(* CODESYS project lab3_pod2.project
   Title: lab2_pod2
   Version: 0.0.0.0
   Author: ichiro

Project tree, tasks and I/O mapping:
  MyController : TM251MESE, Schneider Electric, order no. TM251MESE, version 4.0.6.18
    application Application
      task MAST (cyclic, interval t#1s, priority 15, watchdog 100 ms x 1) calls Task1_1
      global variables GVL
      program TASK1 [ST]
      program TASK2 [ST]
      program TASK3 [ST]
      program TASK5 [ST]
      program TASK4 [ST]
      program Task1_1 [ST]
      Relocation Table
    IO_Bus : IO bus - TM3, Schneider Electric, version 4.0.6.18
      Module_1 : TM3TM3/G, Schneider Electric, order no. TM3TM3/G, version 1.0.1.6
          settings: KPI Configuration.KPI Configuration[0] = 78; KPI Configuration.KPI Configuration[1] = 35; KPI Configuration.KPI Configuration[2] = 48; KPI Configuration.KPI Configuration[3] = 248; KPI Configuration.KPI Configuration[5] = 0; KPI Configuration.KPI Configuration[6] = 112; KPI Configuration.KPI Configuration[7] = 23; KPI Configuration.KPI Configuration[8] = 100; KPI Configuration.KPI Configuration[9] = 0; KPI Configuration.KPI Configuration[16] = 16; KPI Configuration.KPI Configuration[19] = 0; KPI Configuration.KPI Configuration[20] = 192; KPI Configuration.KPI Configuration[21] = 93
          input  temper_in : INT  // IW0
          input  water_in : INT  // IW1
          output motor : INT  // QW0
          input  ibModule_1_IBStatusIW0 : BYTE  // IBStatusIW0
          input  ibModule_1_IBStatusIW1 : BYTE  // IBStatusIW1
          input  ibModule_1_IBStatusQW0 : BYTE  // IBStatusQW0
    COM_Bus : COM bus, Schneider Electric, version 4.0.6.18
    Ethernet_1 : Ethernet Network, Schneider Electric, version 4.0.6.18
      ModbusTCP_Slave_Device : ModbusTCP Slave Device, Schneider Electric, version 3.5.2.6
          input  iwModbusTCP_Slave_Device_Inputs_0 : WORD  // Inputs.Inputs[0]
          input  iwModbusTCP_Slave_Device_Inputs_1 : WORD  // Inputs.Inputs[1]
          input  iwModbusTCP_Slave_Device_Inputs_2 : WORD  // Inputs.Inputs[2]
          input  iwModbusTCP_Slave_Device_Inputs_3 : WORD  // Inputs.Inputs[3]
          input  iwModbusTCP_Slave_Device_Inputs_4 : WORD  // Inputs.Inputs[4]
          input  iwModbusTCP_Slave_Device_Inputs_5 : WORD  // Inputs.Inputs[5]
          input  iwModbusTCP_Slave_Device_Inputs_6 : WORD  // Inputs.Inputs[6]
          input  iwModbusTCP_Slave_Device_Inputs_7 : WORD  // Inputs.Inputs[7]
          input  iwModbusTCP_Slave_Device_Inputs_8 : WORD  // Inputs.Inputs[8]
          input  iwModbusTCP_Slave_Device_Inputs_9 : WORD  // Inputs.Inputs[9]
          output qwModbusTCP_Slave_Device_Outputs_0 : WORD  // Outputs.Outputs[0]
          output qwModbusTCP_Slave_Device_Outputs_1 : WORD  // Outputs.Outputs[1]
          output qwModbusTCP_Slave_Device_Outputs_2 : WORD  // Outputs.Outputs[2]
          output qwModbusTCP_Slave_Device_Outputs_3 : WORD  // Outputs.Outputs[3]
          output qwModbusTCP_Slave_Device_Outputs_4 : WORD  // Outputs.Outputs[4]
          output qwModbusTCP_Slave_Device_Outputs_5 : WORD  // Outputs.Outputs[5]
          output qwModbusTCP_Slave_Device_Outputs_6 : WORD  // Outputs.Outputs[6]
          output qwModbusTCP_Slave_Device_Outputs_7 : WORD  // Outputs.Outputs[7]
          output qwModbusTCP_Slave_Device_Outputs_8 : WORD  // Outputs.Outputs[8]
          output qwModbusTCP_Slave_Device_Outputs_9 : WORD  // Outputs.Outputs[9]
          unmapped channels: Inputs, Outputs
    Ethernet_2 : Device Network, Schneider Electric, version 4.0.6.18
        settings: IPAddress = [10, 77, 70, 112]; SubnetMask = [255, 255, 255, 0]; GatewayAddress = [10, 77, 70, 1]; WebServer = TRUE; FTP Server = TRUE; SoMachine Protocol = TRUE; Modbus Server = TRUE; NetManage Protocol = TRUE; SNMP protocol = TRUE; Enable Routing = FALSE; WebVisu protocol = TRUE; DHCP Server Active = TRUE
      Industrial_Ethernet_Manager : Industrial Ethernet Manager, Schneider Electric, version 1.0.12.20
          settings: BinaryFileSize = 396; Dhcps Host 0.Client Mac Address = [16#0, 16#0, 16#0, 16#0, 16#0]; Dhcps Host 0.Client Device Name = 'DEVICE_1'; Dhcps Host 0.Client IP Address = [10, 77, 70, 111]; Dhcps Host 0.Network Mask = [255, 255, 255, 0]; Dhcps Host 0.Default Gateway = [10, 77, 70, 112]; Dhcps Host 1.Client Mac Address = [16#0, 16#0, 16#0, 16#0, 16#0]; Dhcps Host 2.Client Mac Address = [16#0, 16#0, 16#0, 16#0, 16#0]; Dhcps Host 3.Client Mac Address = [16#0, 16#0, 16#0, 16#0, 16#0]; Dhcps Host 4.Client Mac Address = [16#0, 16#0, 16#0, 16#0, 16#0]; Dhcps Host 5.Client Mac Address = [16#0, 16#0, 16#0, 16#0, 16#0]; Dhcps Host 6.Client Mac Address = [16#0, 16#0, 16#0, 16#0, 16#0]; Dhcps Host 7.Client Mac Address = [16#0, 16#0, 16#0, 16#0, 16#0]; Dhcps Host 8.Client Mac Address = [16#0, 16#0, 16#0, 16#0, 16#0]; Dhcps Host 9.Client Mac Address = [16#0, 16#0, 16#0, 16#0, 16#0]; Dhcps Host 10.Client Mac Address = [16#0, 16#0, 16#0, 16#0, 16#0]; Dhcps Host 11.Client Mac Address = [16#0, 16#0, 16#0, 16#0, 16#0]; Dhcps Host 12.Client Mac Address = [16#0, 16#0, 16#0, 16#0, 16#0]; Dhcps Host 13.Client Mac Address = [16#0, 16#0, 16#0, 16#0, 16#0]; Dhcps Host 14.Client Mac Address = [16#0, 16#0, 16#0, 16#0, 16#0]; Dhcps Host 15.Client Mac Address = [16#0, 16#0, 16#0, 16#0, 16#0]; Dhcps Host 16.Client Mac Address = [16#0, 16#0, 16#0, 16#0, 16#0]; Dhcps Host 17.Client Mac Address = [16#0, 16#0, 16#0, 16#0, 16#0]; Dhcps Host 18.Client Mac Address = [16#0, 16#0, 16#0, 16#0, 16#0]; Dhcps Host 19.Client Mac Address = [16#0, 16#0, 16#0, 16#0, 16#0]; Dhcps Host 20.Client Mac Address = [16#0, 16#0, 16#0, 16#0, 16#0]; Dhcps Host 21.Client Mac Address = [16#0, 16#0, 16#0, 16#0, 16#0]; Dhcps Host 22.Client Mac Address = [16#0, 16#0, 16#0, 16#0, 16#0]; Dhcps Host 23.Client Mac Address = [16#0, 16#0, 16#0, 16#0, 16#0]; Dhcps Host 24.Client Mac Address = [16#0, 16#0, 16#0, 16#0, 16#0]; Dhcps Host 25.Client Mac Address = [16#0, 16#0, 16#0, 16#0, 16#0]; Dhcps Host 26.Client Mac Address = [16#0, 16#0, 16#0, 16#0, 16#0]; Dhcps Host 27.Client Mac Address = [16#0, 16#0, 16#0, 16#0, 16#0]; Dhcps Host 28.Client Mac Address = [16#0, 16#0, 16#0, 16#0, 16#0]; Dhcps Host 29.Client Mac Address = [16#0, 16#0, 16#0, 16#0, 16#0]; Dhcps Host 30.Client Mac Address = [16#0, 16#0, 16#0, 16#0, 16#0]; Dhcps Host 31.Client Mac Address = [16#0, 16#0, 16#0, 16#0, 16#0]; Dhcps Host 32.Client Mac Address = [16#0, 16#0, 16#0, 16#0, 16#0]; Dhcps Host 33.Client Mac Address = [16#0, 16#0, 16#0, 16#0, 16#0]; Dhcps Host 34.Client Mac Address = [16#0, 16#0, 16#0, 16#0, 16#0];
            Dhcps Host 35.Client Mac Address = [16#0, 16#0, 16#0, 16#0, 16#0]; Dhcps Host 36.Client Mac Address = [16#0, 16#0, 16#0, 16#0, 16#0]; Dhcps Host 37.Client Mac Address = [16#0, 16#0, 16#0, 16#0, 16#0]; Dhcps Host 38.Client Mac Address = [16#0, 16#0, 16#0, 16#0, 16#0]; Dhcps Host 39.Client Mac Address = [16#0, 16#0, 16#0, 16#0, 16#0]; Dhcps Host 40.Client Mac Address = [16#0, 16#0, 16#0, 16#0, 16#0]; Dhcps Host 41.Client Mac Address = [16#0, 16#0, 16#0, 16#0, 16#0]; Dhcps Host 42.Client Mac Address = [16#0, 16#0, 16#0, 16#0, 16#0]; Dhcps Host 43.Client Mac Address = [16#0, 16#0, 16#0, 16#0, 16#0]; Dhcps Host 44.Client Mac Address = [16#0, 16#0, 16#0, 16#0, 16#0]; Dhcps Host 45.Client Mac Address = [16#0, 16#0, 16#0, 16#0, 16#0]; Dhcps Host 46.Client Mac Address = [16#0, 16#0, 16#0, 16#0, 16#0]; Dhcps Host 47.Client Mac Address = [16#0, 16#0, 16#0, 16#0, 16#0]; Dhcps Host 48.Client Mac Address = [16#0, 16#0, 16#0, 16#0, 16#0]; Dhcps Host 49.Client Mac Address = [16#0, 16#0, 16#0, 16#0, 16#0]; Dhcps Host 50.Client Mac Address = [16#0, 16#0, 16#0, 16#0, 16#0]; Dhcps Host 51.Client Mac Address = [16#0, 16#0, 16#0, 16#0, 16#0]; Dhcps Host 52.Client Mac Address = [16#0, 16#0, 16#0, 16#0, 16#0]; Dhcps Host 53.Client Mac Address = [16#0, 16#0, 16#0, 16#0, 16#0]; Dhcps Host 54.Client Mac Address = [16#0, 16#0, 16#0, 16#0, 16#0]; Dhcps Host 55.Client Mac Address = [16#0, 16#0, 16#0, 16#0, 16#0]; Dhcps Host 56.Client Mac Address = [16#0, 16#0, 16#0, 16#0, 16#0]; Dhcps Host 57.Client Mac Address = [16#0, 16#0, 16#0, 16#0, 16#0]; Dhcps Host 58.Client Mac Address = [16#0, 16#0, 16#0, 16#0, 16#0]; Dhcps Host 59.Client Mac Address = [16#0, 16#0, 16#0, 16#0, 16#0]; Dhcps Host 60.Client Mac Address = [16#0, 16#0, 16#0, 16#0, 16#0]; Dhcps Host 61.Client Mac Address = [16#0, 16#0, 16#0, 16#0, 16#0]; Dhcps Host 62.Client Mac Address = [16#0, 16#0, 16#0, 16#0, 16#0]; Dhcps Host 63.Client Mac Address = [16#0, 16#0, 16#0, 16#0, 16#0]; Dhcps Host 64.Client Mac Address = [16#0, 16#0, 16#0, 16#0, 16#0]; Dhcps Host 65.Client Mac Address = [16#0, 16#0, 16#0, 16#0, 16#0]; Dhcps Host 66.Client Mac Address = [16#0, 16#0, 16#0, 16#0, 16#0]; Dhcps Host 67.Client Mac Address = [16#0, 16#0, 16#0, 16#0, 16#0]; Dhcps Host 68.Client Mac Address = [16#0, 16#0, 16#0, 16#0, 16#0]; Dhcps Host 69.Client Mac Address = [16#0, 16#0, 16#0, 16#0, 16#0]; Dhcps Host 70.Client Mac Address = [16#0, 16#0, 16#0, 16#0, 16#0]; Dhcps Host 71.Client Mac Address = [16#0, 16#0, 16#0, 16#0, 16#0]; Dhcps Host 72.Client Mac Address = [16#0, 16#0, 16#0, 16#0, 16#0]; Dhcps Host 73.Client Mac Address = [16#0, 16#0, 16#0, 16#0, 16#0]; Dhcps Host 74.Client Mac Address = [16#0, 16#0, 16#0, 16#0, 16#0];
            Dhcps Host 75.Client Mac Address = [16#0, 16#0, 16#0, 16#0, 16#0]; Dhcps Host 76.Client Mac Address = [16#0, 16#0, 16#0, 16#0, 16#0]; Dhcps Host 77.Client Mac Address = [16#0, 16#0, 16#0, 16#0, 16#0]; Dhcps Host 78.Client Mac Address = [16#0, 16#0, 16#0, 16#0, 16#0]; Dhcps Host 79.Client Mac Address = [16#0, 16#0, 16#0, 16#0, 16#0]; Dhcps Host 80.Client Mac Address = [16#0, 16#0, 16#0, 16#0, 16#0]; Dhcps Host 81.Client Mac Address = [16#0, 16#0, 16#0, 16#0, 16#0]; Dhcps Host 82.Client Mac Address = [16#0, 16#0, 16#0, 16#0, 16#0]; Dhcps Host 83.Client Mac Address = [16#0, 16#0, 16#0, 16#0, 16#0]; Dhcps Host 84.Client Mac Address = [16#0, 16#0, 16#0, 16#0, 16#0]; Dhcps Host 85.Client Mac Address = [16#0, 16#0, 16#0, 16#0, 16#0]; Dhcps Host 86.Client Mac Address = [16#0, 16#0, 16#0, 16#0, 16#0]; Dhcps Host 87.Client Mac Address = [16#0, 16#0, 16#0, 16#0, 16#0]; Dhcps Host 88.Client Mac Address = [16#0, 16#0, 16#0, 16#0, 16#0]; Dhcps Host 89.Client Mac Address = [16#0, 16#0, 16#0, 16#0, 16#0]; Dhcps Host 90.Client Mac Address = [16#0, 16#0, 16#0, 16#0, 16#0]; Dhcps Host 91.Client Mac Address = [16#0, 16#0, 16#0, 16#0, 16#0]; Dhcps Host 92.Client Mac Address = [16#0, 16#0, 16#0, 16#0, 16#0]; Dhcps Host 93.Client Mac Address = [16#0, 16#0, 16#0, 16#0, 16#0]; Dhcps Host 94.Client Mac Address = [16#0, 16#0, 16#0, 16#0, 16#0]; Dhcps Host 95.Client Mac Address = [16#0, 16#0, 16#0, 16#0, 16#0]; Dhcps Host 96.Client Mac Address = [16#0, 16#0, 16#0, 16#0, 16#0]; Dhcps Host 97.Client Mac Address = [16#0, 16#0, 16#0, 16#0, 16#0]; Dhcps Host 98.Client Mac Address = [16#0, 16#0, 16#0, 16#0, 16#0]; Dhcps Host 99.Client Mac Address = [16#0, 16#0, 16#0, 16#0, 16#0]; Dhcps Host 100.Client Mac Address = [16#0, 16#0, 16#0, 16#0, 16#0]; Dhcps Host 101.Client Mac Address = [16#0, 16#0, 16#0, 16#0, 16#0]; Dhcps Host 102.Client Mac Address = [16#0, 16#0, 16#0, 16#0, 16#0]; Dhcps Host 103.Client Mac Address = [16#0, 16#0, 16#0, 16#0, 16#0]; Dhcps Host 104.Client Mac Address = [16#0, 16#0, 16#0, 16#0, 16#0]; Dhcps Host 105.Client Mac Address = [16#0, 16#0, 16#0, 16#0, 16#0]; Dhcps Host 106.Client Mac Address = [16#0, 16#0, 16#0, 16#0, 16#0]; Dhcps Host 107.Client Mac Address = [16#0, 16#0, 16#0, 16#0, 16#0]; Dhcps Host 108.Client Mac Address = [16#0, 16#0, 16#0, 16#0, 16#0]; Dhcps Host 109.Client Mac Address = [16#0, 16#0, 16#0, 16#0, 16#0]; Dhcps Host 110.Client Mac Address = [16#0, 16#0, 16#0, 16#0, 16#0]; Dhcps Host 111.Client Mac Address = [16#0, 16#0, 16#0, 16#0, 16#0]; Dhcps Host 112.Client Mac Address = [16#0, 16#0, 16#0, 16#0, 16#0]; Dhcps Host 113.Client Mac Address = [16#0, 16#0, 16#0, 16#0, 16#0]; Dhcps Host 114.Client Mac Address = [16#0, 16#0, 16#0, 16#0, 16#0];
            Dhcps Host 115.Client Mac Address = [16#0, 16#0, 16#0, 16#0, 16#0]; Dhcps Host 116.Client Mac Address = [16#0, 16#0, 16#0, 16#0, 16#0]; Dhcps Host 117.Client Mac Address = [16#0, 16#0, 16#0, 16#0, 16#0]; Dhcps Host 118.Client Mac Address = [16#0, 16#0, 16#0, 16#0, 16#0]; Dhcps Host 119.Client Mac Address = [16#0, 16#0, 16#0, 16#0, 16#0]; Dhcps Host 120.Client Mac Address = [16#0, 16#0, 16#0, 16#0, 16#0]; Dhcps Host 121.Client Mac Address = [16#0, 16#0, 16#0, 16#0, 16#0]; Dhcps Host 122.Client Mac Address = [16#0, 16#0, 16#0, 16#0, 16#0]; Dhcps Host 123.Client Mac Address = [16#0, 16#0, 16#0, 16#0, 16#0]; Dhcps Host 124.Client Mac Address = [16#0, 16#0, 16#0, 16#0, 16#0]; Dhcps Host 125.Client Mac Address = [16#0, 16#0, 16#0, 16#0, 16#0]; Dhcps Host 126.Client Mac Address = [16#0, 16#0, 16#0, 16#0, 16#0]; Dhcps Host 127.Client Mac Address = [16#0, 16#0, 16#0, 16#0, 16#0]; Dhcps Host 128.Client Mac Address = [16#0, 16#0, 16#0, 16#0, 16#0]; serialized Values = 6924ca37-4fff-47b2-bdf6-b3d002c8f643=0|
          unmapped channels: Global Status, Healthbit 0, Healthbit 1, Healthbit 2, Healthbit 3
        Generic_Modbus_TCP_Slave : Generic Modbus TCP Slave, Schneider Electric, version 1.0.2.21
            settings: Unit-ID = 248; IPAddress = [10, 77, 70, 111]; SubnetMask = [0, 0, 0, 0]; DeviceName = 'DEVICE_1'; Channel_cmd.Channel ID = 0; Channel_cmd.Unit-ID = 1; Channel_cmd.Repetition Rate = 20; Channel_cmd.Function Code = 23; Channel_cmd.Read Offset = 16#2135; Channel_cmd.Read Length = 1; Channel_cmd.Write Offset = 16#2135; Channel_cmd.Write Length = 1; Channel_lfr.Channel ID = 1; Channel_lfr.Unit-ID = 1; Channel_lfr.Repetition Rate = 20; Channel_lfr.Function Code = 23; Channel_lfr.Read Offset = 16#2136; Channel_lfr.Read Length = 1; Channel_lfr.Write Offset = 16#2136; Channel_lfr.Write Length = 1
            output Application.cmd_reg : WORD  // Channel_cmd
            output Application.lft_reg : WORD  // Channel_lfr
            unmapped channels: Channel_cmd, Channel_lfr
    Serial_Line_1 : Serial line, Schneider Electric, version 4.0.6.18
      SoMachine_Network_Manager : SoMachine-Network Manager, Schneider Electric, version 4.0.0.2
*)

// MyController/Application/GVL
VAR_GLOBAL
	foo: INT;
	cmd_reg: WORD := 0;
	lft_reg: INT := 0;
END_VAR

// MyController/Application/Task1_1
PROGRAM Task1_1
VAR 
	counter : INT := 0;
END_VAR

lft_reg := counter * 20;
cmd_reg := 1;
IF (counter = 30) THEN
	counter := 0;
ELSE
	counter := counter + 1;
END_IF

END_PROGRAM

// MyController/Application/TASK1
PROGRAM TASK1
VAR
	timer:TP;
	start:BOOL;
	
END_VAR

timer(IN:=start,PT:=T#30S);
IF start AND timer.Q THEN 
	motor:=12000;
ELSIF start AND NOT timer.Q THEN
	motor:=0;
END_IF

END_PROGRAM

// MyController/Application/TASK2
PROGRAM TASK2
VAR
	start:BOOL;
END_VAR

IF water_in >= 80 THEN
	motor:=12000;
ELSIF water_in <= 50 THEN
	motor:=0;
END_IF

END_PROGRAM

// MyController/Application/TASK3
PROGRAM TASK3
VAR
	PROP:REAL;
END_VAR

PROP:=(TEMPER_IN-230.0)/(340.0-230.0);
IF PROP > 0 THEN
MOTOR:=REAL_TO_INT(PROP*24000);
END_IF

END_PROGRAM

// MyController/Application/TASK5
PROGRAM TASK5
VAR
	PROP:REAL;
END_VAR

PROP:=(TEMPER_IN-230.0)/(340.0-230.0);
IF PROP > 0 AND WATER_IN < 80 THEN
	MOTOR:=REAL_TO_INT(PROP*24000);
ELSIF PROP > 0 AND WATER_IN >= 80 THEN
	MOTOR:=REAL_TO_INT((PROP*24000)/2);
END_IF

END_PROGRAM

// MyController/Application/TASK4
PROGRAM TASK4
VAR
	timer:TP;
	start:BOOL;
END_VAR

timer(IN:=start,PT:=T#30S);
IF start AND timer.ET<=T#10S THEN 
	motor:=3000;
ELSIF start AND timer.ET<T#30S THEN
	motor:=6000;
ELSE
	MOTOR:=0;
END_IF

END_PROGRAM
